FUNCTION_BLOCK FB_DigitalSensor_Test EXTENDS TcUnit.FB_TestSuite
VAR
    // The actual sensor we are going to test
    Sensor : FB_DigitalSensor;
END_VAR

END_FUNCTION_BLOCK

(* stored: Version 1.1.0.1
   POU FB_DigitalSensor_Test: Id {debe6a43-ef40-42e3-9cbd-7e66ae9fa4e4}, SpecialFunc None *)
